(* PLC project GenTraj, Lolitech GenTraj 1.0 *)
(* stored: creationDateTime 2009-01-13T12:15:00, modificationDateTime 2009-01-14T20:10:13 *)

FUNCTION_BLOCK GenTraj
  VAR_INPUT
    Period : REAL;
    Gmvt : REAL;
    Vmvt : REAL;
    P0 : REAL;
    V0 : REAL;
    Pf : REAL;
    Vf : REAL;
  END_VAR
  VAR_OUTPUT
    Pn : REAL;
    Vn : REAL;
    Gn : REAL;
  END_VAR
  VAR
    P : REAL;
    F : REAL;
    Ps2 : REAL;
    Fs3 : REAL;
    delta : REAL;
    Va : REAL;
    Vb : REAL;
    Vaut : REAL;
  END_VAR

IF Period <> P THEN
  P := Period;
  F := 1.0 / P;
  Ps2 := P / 2.0;
  Fs3 := F / 3.0;
END_IF;

IF Pf <> Pn THEN
  delta := Pf - P0 - V0 * P;
  
  Va := SQRT(ABS(2.0 * Gmvt * delta) + Vf * Vf);
  Vb := Vf + delta * Fs3;

  IF Va > ABS(Vb) THEN
    Vaut := MIN(ABS(Vb), Vmvt);
    IF Vb < 0.0 THEN
      Vaut := -Vaut;
    END_IF;
  ELSE
    Vaut := MIN(Va, Vmvt);
    IF Pf < P0 THEN
      Vaut := -Vaut;
    END_IF;    
  END_IF;

  Gn := MIN(ABS((Vaut - V0) * F), Gmvt);
  IF Vaut < V0 THEN
    Gn := -Gn;
  END_IF;

END_IF;

Vn := V0 + Gn * P;

Pn := P0 + (Vn + V0) * Ps2;

IF (P0 >= Pf) <> (Pn >= Pf) AND Vf <> 0.0 THEN
  Pn := Pf;
END_IF;


          
END_FUNCTION_BLOCK

PROGRAM TestMotion
  VAR
    GO : BOOL := TRUE;
    TRIG : BOOL;
    GenTraj1 : GenTraj;
    py_eval : python_eval;
    RS1 : RS;
  END_VAR
  VAR  (* added by the conversion: wires and edge detectors of the diagram *)
    _NOT15_OUT : BOOL;
  END_VAR

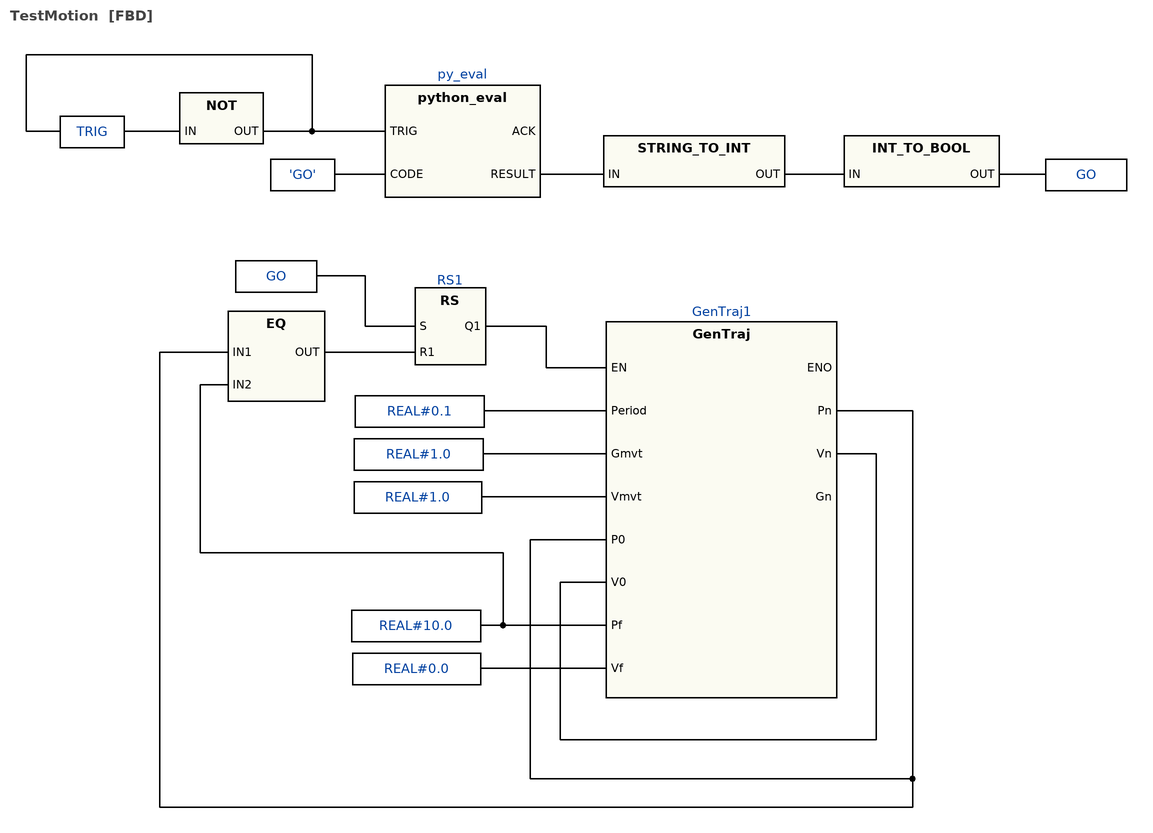
(* FBD diagram, written out as Structured Text *)
_NOT15_OUT := NOT TRIG;
TRIG := _NOT15_OUT;
py_eval(TRIG := _NOT15_OUT, CODE := 'GO');
GO := INT_TO_BOOL(STRING_TO_INT(py_eval.RESULT));
GenTraj1(EN := RS1.Q1, Period := REAL#0.1, Gmvt := REAL#1.0, Vmvt := REAL#1.0, P0 := GenTraj1.Pn, V0 := GenTraj1.Vn, Pf := REAL#10.0, Vf := REAL#0.0);
RS1(S := GO, R1 := GenTraj1.Pn = REAL#10.0);
END_PROGRAM

CONFIGURATION config
  RESOURCE ress ON PLC
    TASK MAIN_TASK(INTERVAL := 00:00:00.100000, PRIORITY := 0);
    PROGRAM MAIN_INSTANCE WITH MAIN_TASK : TestMotion;
  END_RESOURCE
END_CONFIGURATION
